(* CODESYS project MID_GPS_GPRS_Demo.project

Project tree, tasks and I/O mapping:
  Device : Changsha Xiangji-ARM Cortex A9(xilinx zynq7000)-linux, Changsha Xiangji Hiden Technology Co.Ltd, version 3.5.10.20
    application Application
      libraries: Standard, * (System); CAA DTUtil Extern, * (CAA Technical Workgroup); CAA SerialCom, * (CAA Technical Workgroup); CAA Types Extern, * (CAA Technical Workgroup); AC_Persistence, * (3S - Smart Software Solutions GmbH)
      task MainTask (cyclic, interval 4 ms, priority 1) calls MC20_serial, PLC_PRG
      task VISU_TASK (cyclic, interval 100 ms, priority 31) calls VisuElems.Visu_Prg
      program PLC_PRG [ST]
      global variables GVL
      program MC20_serial [ST]
      visualisation Main_test_Visua
    SoftMotion General Axis Pool
  text list GlobalTextList
*)

// Device/Application/GVL
{attribute 'qualified_only'}
{attribute 'qualified_only'}

VAR_GLOBAL

	NewDT : DT;
	NewDTS : STRING;
	NewDTSZH : STRING;
	cmdSend:BOOL := FALSE;
	recvOk:BOOL := FALSE;

	send_serial :BYTE := 0;

	
END_VAR

// Device/Application/MC20_serial
PROGRAM MC20_serial
VAR
	Com1Params: 			ARRAY [1..7] OF COM.PARAMETER;	(* Settings to communicate with the COM Port *)
	hCom: 					CAA.HANDLE;
	ComOpen: 				COM.Open;
	ComClose: 				COM.Close;
	ComWrite: 				COM.Write;
	ComRead: 				COM.Read;	
	//Writebuffer: 			STRING:= 'Hello! zhouqin';

	Snd_Cnt:				CAA.SIZE;

	Rcv_Cnt: 				CAA.SIZE;
	xCom1CloseError: 		BOOL;
	xCom1WriteError: 		BOOL;
	xCom1ReadError: 		BOOL;
	xError:					BOOL;
	
	uiComState: INT := 0;
	uiComState_MC20: INT := 0;
	ComID_MC20:USINT:=3;//串口号为4

	cmdSend:BOOL := FALSE;
	COMWritebufsum_MC20: 	    STRING(200):='';
	COMReadbufsum_MC20: 			STRING(200);
	ton2:TON;
	size:CAA.SIZE;
	
	at_ask_buffer1 :STRING(1000);
	at_ask_buffer2 :STRING(1000);
	at_ask_buffer3 :STRING(1000);
	at_ask_buffer4 :STRING(1000);
	at_ask_buffer5:STRING(1000);
	at_ask_buffer6 :STRING(1000);
	
	
	bit_start:INT;
	bit_end:INT;
	bit_start1:INT;
	bit_end1:INT;
	jd_info:STRING;
	wd_info:STRING;
	jd:REAL;
	wd:REAL;
	R_TIME:TIME;
	
END_VAR


CASE uiComState_MC20 OF
	0:
	Com1Params[1].udiParameterId := COM.CAA_Parameter_Constants.udiPort;
	Com1Params[1].udiValue := ComID_MC20; 
	Com1Params[2].udiParameterId := COM.CAA_Parameter_Constants.udiBaudrate;
	Com1Params[2].udiValue := 115200;
	Com1Params[3].udiParameterId := COM.CAA_Parameter_Constants.udiParity;
	Com1Params[3].udiValue := INT_TO_UINT(COM.PARITY.NONE);
	Com1Params[4].udiParameterId := COM.CAA_Parameter_Constants.udiStopBits;
	Com1Params[4].udiValue := INT_TO_UINT(COM.STOPBIT.ONESTOPBIT);
	Com1Params[5].udiParameterId := COM.CAA_Parameter_Constants.udiTimeout;
	Com1Params[5].udiValue := 0;
	Com1Params[6].udiParameterId := COM.CAA_Parameter_Constants.udiByteSize;
	Com1Params[6].udiValue := 8;
	Com1Params[7].udiParameterId := COM.CAA_Parameter_Constants.udiBinary;
	Com1Params[7].udiValue := 0;					
	ComOpen(xExecute := TRUE, usiListLength:=UINT_TO_USINT(SIZEOF(Com1Params)/SIZEOF(COM.PARAMETER)),pParameterList:= ADR(Com1Params),hCom=> hCom);			
	IF ComOpen.xError THEN
		uiComState_MC20 := 32767;
	ELSIF ComOpen.xDone THEN
		uiComState_MC20 := 1;
	END_IF
	
	1:
	COMWritebufsum_MC20:='AT$r';//发送AT指令，测试串口和MC20是否正常通信
	gvl.cmdSend:=TRUE;
	IF gvl.cmdSend  THEN
		ComWrite(xExecute := TRUE,hCom:= hCom,pBuffer:= ADR(COMWritebufsum_MC20),szSize:= ANY_TO_UDINT(len(COMWritebufsum_MC20)));		
		IF ComWrite.xError THEN
			uiComState_MC20 := 32767;
		END_IF
		IF ComWrite.xDone THEN		
			ComWrite(xExecute := FALSE);
			uiComState_MC20 := 2;
			gvl.send_serial := gvl.send_serial + 1;
			gvl.cmdSend := FALSE;
			gvl.recvOk := FALSE;
		END_IF
	END_IF
	
   2:
	TON2(IN:=TRUE,PT:=T#200MS);
		IF TON2.Q=TRUE THEN
	        	ComRead(xExecute := FALSE,hCom:= hCom, pBuffer:= ADR(COMReadbufsum_MC20), szBuffer:= SIZEOF(COMReadbufsum_MC20));	
	            COMReadbufsum_MC20:='';	
				uiComState_MC20 := 3;	
				TON2(IN:=FALSE,PT:=T#200MS);
		END_IF
	
	3:
	ComRead(xExecute := TRUE,hCom:= hCom, pBuffer:= ADR(COMReadbufsum_MC20), szBuffer:= SIZEOF(COMReadbufsum_MC20));
	IF ComRead.xError THEN
		uiComState_MC20 := 32767;
	END_IF	

    IF ComRead.xDone THEN
	  at_ask_buffer1:=COMReadbufsum_MC20;
	  uiComState_MC20 := 4;	
	END_IF


	4: 
	COMWritebufsum_MC20:='AT+QGNSSC=1$r';//发送AT指令，启动模块的GPS功能
	gvl.cmdSend:=TRUE;
	IF gvl.cmdSend  THEN
		ComWrite(xExecute := TRUE,hCom:= hCom,pBuffer:= ADR(COMWritebufsum_MC20),szSize:= ANY_TO_UDINT(len(COMWritebufsum_MC20)));		
		IF ComWrite.xError THEN
			uiComState_MC20 := 32767;
		END_IF
		IF ComWrite.xDone THEN		
			ComWrite(xExecute := FALSE);
			uiComState_MC20 := 5;
			gvl.send_serial := gvl.send_serial + 1;
			gvl.cmdSend := FALSE;
			gvl.recvOk := FALSE;
		END_IF
	END_IF
	
  5:
	TON2(IN:=TRUE,PT:=T#200MS);
		IF TON2.Q=TRUE THEN
                ComRead(xExecute := FALSE,hCom:= hCom, pBuffer:= ADR(COMReadbufsum_MC20), szBuffer:= SIZEOF(COMReadbufsum_MC20));		
	            COMReadbufsum_MC20:='';	
                uiComState_MC20 := 6;
				TON2(IN:=FALSE,PT:=T#200MS);
		END_IF
	
	6: 
	ComRead(xExecute := TRUE,hCom:= hCom, pBuffer:= ADR(COMReadbufsum_MC20), szBuffer:= SIZEOF(COMReadbufsum_MC20));
	IF ComRead.xError THEN
		uiComState_MC20 := 32767;
	END_IF

    IF ComRead.xDone THEN
	  at_ask_buffer2:=COMReadbufsum_MC20;
	  uiComState_MC20 := 7;	
	END_IF
	
	 7:

      uiComState_MC20 := 8;
	
	
	
	
	8:  
	COMWritebufsum_MC20:='AT+QGNSSRD="NMEA/RMC"$r';//发送AT指令，查询获取的经纬度
	gvl.cmdSend:=TRUE;
	IF gvl.cmdSend  THEN
		ComWrite(xExecute := TRUE,hCom:= hCom,pBuffer:= ADR(COMWritebufsum_MC20),szSize:= ANY_TO_UDINT(len(COMWritebufsum_MC20)));		
		IF ComWrite.xError THEN
			uiComState_MC20 := 32767;
		END_IF
		IF ComWrite.xDone THEN		
			ComWrite(xExecute := FALSE);
			uiComState_MC20 := 9;
			gvl.send_serial := gvl.send_serial + 1;
			gvl.cmdSend := FALSE;
			gvl.recvOk := FALSE;
		END_IF
	END_IF
	
	9:
	TON2(IN:=TRUE,PT:=T#200MS);
		IF TON2.Q=TRUE THEN
				ComRead(xExecute := FALSE,hCom:= hCom, pBuffer:= ADR(COMReadbufsum_MC20), szBuffer:= SIZEOF(COMReadbufsum_MC20));	//给xExecute制造一个上升沿，读串口命令才能被调用一次
	            COMReadbufsum_MC20:='';	
                uiComState_MC20 := 10;
				TON2(IN:=FALSE,PT:=T#200MS);
		END_IF
	
	10:
	ComRead(xExecute := TRUE,hCom:= hCom, pBuffer:= ADR(COMReadbufsum_MC20), szBuffer:= SIZEOF(COMReadbufsum_MC20));
	IF ComRead.xError THEN
		uiComState_MC20 := 32767;
	END_IF
    IF ComRead.xDone THEN
	  at_ask_buffer3:=COMReadbufsum_MC20;
	//解析经纬度信息，正确的 回复格式为消息：+QGNSSRD: $GNRMC,023740.000,A,2813.8648,N,11324.8867,E,0.42,353.49,020419,,,A*7C
   bit_start:=FIND( at_ask_buffer3,',A');
   bit_end:=FIND( at_ask_buffer3,',N');//读换行符的位置
   jd_info:=mid( at_ask_buffer3,bit_end-bit_start-1,bit_start+3);
   jd:=ANY_TO_REAL(jd_info)/100;
   bit_start1:=FIND( at_ask_buffer3,'N,');
   bit_end1:=FIND( at_ask_buffer3,',E');//读换行符的位置
   wd_info:=mid( at_ask_buffer3,bit_end1-bit_start1-1,bit_start1+2);
   wd:=ANY_TO_REAL(wd_info)/100;  
	 IF  jd=0 OR wd=0 THEN
		 uiComState_MC20 := 8;
     ELSE
		  uiComState_MC20 := 11;
	 END_IF
	  
	 	
	END_IF
	
	11:  
	COMWritebufsum_MC20:='AT+QNITZ=1$r';	//启用同步网络时间
	gvl.cmdSend:=TRUE;
	IF gvl.cmdSend  THEN
		ComWrite(xExecute := TRUE,hCom:= hCom,pBuffer:= ADR(COMWritebufsum_MC20),szSize:= ANY_TO_UDINT(len(COMWritebufsum_MC20)));		
		IF ComWrite.xError THEN
			uiComState_MC20 := 32767;
		END_IF
		IF ComWrite.xDone THEN		
			ComWrite(xExecute := FALSE);
			uiComState_MC20 := 12;
			gvl.send_serial := gvl.send_serial + 1;
			gvl.cmdSend := FALSE;
			gvl.recvOk := FALSE;
		END_IF
	END_IF
	
	12:
	TON2(IN:=TRUE,PT:=T#200MS);
		IF TON2.Q=TRUE THEN
				ComRead(xExecute := FALSE,hCom:= hCom, pBuffer:= ADR(COMReadbufsum_MC20), szBuffer:= SIZEOF(COMReadbufsum_MC20));	//给xExecute制造一个上升沿，读串口命令才能被调用一次
	            COMReadbufsum_MC20:='';	
                uiComState_MC20 := 13;
				TON2(IN:=FALSE,PT:=T#200MS);
		END_IF
	
	13:
	ComRead(xExecute := TRUE,hCom:= hCom, pBuffer:= ADR(COMReadbufsum_MC20), szBuffer:= SIZEOF(COMReadbufsum_MC20));
	IF ComRead.xError THEN
		uiComState_MC20 := 32767;
	END_IF
    IF ComRead.xDone THEN
	  at_ask_buffer4:=COMReadbufsum_MC20;
	  uiComState_MC20 := 14;	
	END_IF
	
    14:  
	COMWritebufsum_MC20:='AT+CCLK?$r';	//启获取模块的实时时钟
	gvl.cmdSend:=TRUE;
	IF gvl.cmdSend  THEN
		ComWrite(xExecute := TRUE,hCom:= hCom,pBuffer:= ADR(COMWritebufsum_MC20),szSize:= ANY_TO_UDINT(len(COMWritebufsum_MC20)));		
		IF ComWrite.xError THEN
			uiComState_MC20 := 32767;
		END_IF
		IF ComWrite.xDone THEN		
			ComWrite(xExecute := FALSE);
			uiComState_MC20 := 15;
			gvl.send_serial := gvl.send_serial + 1;
			gvl.cmdSend := FALSE;
			gvl.recvOk := FALSE;
		END_IF
	END_IF
	
	15:
	TON2(IN:=TRUE,PT:=T#200MS);
		IF TON2.Q=TRUE THEN
				ComRead(xExecute := FALSE,hCom:= hCom, pBuffer:= ADR(COMReadbufsum_MC20), szBuffer:= SIZEOF(COMReadbufsum_MC20));	//给xExecute制造一个上升沿，读串口命令才能被调用一次
	            COMReadbufsum_MC20:='';	
                uiComState_MC20 := 16;
				TON2(IN:=FALSE,PT:=T#200MS);
		END_IF
	
	16:
	ComRead(xExecute := TRUE,hCom:= hCom, pBuffer:= ADR(COMReadbufsum_MC20), szBuffer:= SIZEOF(COMReadbufsum_MC20));
	IF ComRead.xError THEN
		uiComState_MC20 := 32767;
	END_IF
    IF ComRead.xDone THEN
	  at_ask_buffer5:=COMReadbufsum_MC20;
      GVL.NewDTS:=MID(at_ask_buffer5,17,20);
	  
	  gvl.NewDTSZH:=CONCAT('DT#20',left(GVL.NewDTS,2));
	  gvl.NewDTSZH:=CONCAT(gvl.NewDTSZH,'-');	  
	  gvl.NewDTSZH:=CONCAT(gvl.NewDTSZH,mid(GVL.NewDTS,2,4));	 
      gvl.NewDTSZH:=CONCAT(gvl.NewDTSZH,'-');	
	  gvl.NewDTSZH:=CONCAT(gvl.NewDTSZH,mid(GVL.NewDTS,2,7));	
      gvl.NewDTSZH:=CONCAT(gvl.NewDTSZH,'-');	
 	  gvl.NewDTSZH:=CONCAT(gvl.NewDTSZH,mid(GVL.NewDTS,8,10));		  
	  GVL.NewDT:=ANY_TO_DT(gvl.NewDTSZH);
	  PLC_PRG.dtu_set_dt_fb.dtDateAndTime := STRING_TO_DT(gvl.NewDTSZH);
	  PLC_PRG.dtu_set_dt_fb(xExecute := FALSE);
	  PLC_PRG.dtu_set_dt_fb.xExecute := TRUE;
	  
	  
	  uiComState_MC20 := 32767;	
	END_IF
	255:
	
	32767:	
END_CASE

END_PROGRAM

// Device/Application/PLC_PRG
PROGRAM PLC_PRG
VAR
	ton1:TON;
	dtu_get_dt_fb:dtu.GetDateAndTime;
	Mydt:DT;
	MydtS:STRING;
END_VAR
VAR_INPUT	
	dtu_set_dt_fb: dtu.SetDateAndTime;
END_VAR



//时钟走时
    dtu_set_dt_fb();//将MC20读到的时钟同步到系统时钟里面去
	TON1(IN:=TRUE,PT:=T#1S);//系统时钟走时，每秒读一次系统时钟
		IF TON1.Q=TRUE THEN
				Mydt:=GETdatetime();		
				MydtS:=ANY_TO_STRING(Mydt);
				TON1(IN:=FALSE,PT:=T#1S);
		END_IF

END_PROGRAM

// Device/Application/Main_test_Visua
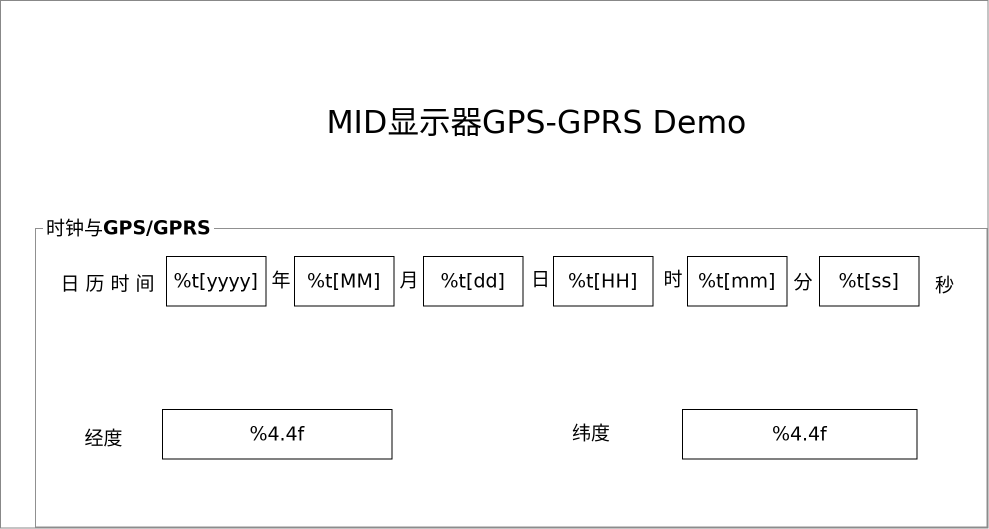
VISUALIZATION Main_test_Visua  // 989x529
    GroupBox (35,220 952x307), "时钟与GPS/GPRS"
        Rectangle (127,189 230x50), "%4.4f", text variable: MC20_serial.jd
        Rectangle (647,189 235x50), "%4.4f", text variable: MC20_serial.wd
        Label (507,186 98x54), "纬度"
        Label (12,188 113x60), "经度"
        Rectangle (784,36 100x50), "%t[ss]", text variable: PLC_PRG.MydtS
        Label (742,29 52x66), "分"
        Rectangle (652,36 100x50), "%t[mm]", text variable: PLC_PRG.MydtS
        Label (607,26 62x66), "时"
        Label (473,25 65x68), "日"
        Label (219,25 54x70), "年"
        Label (343,23 62x74), "月"
        Rectangle (518,36 100x50), "%t[HH]", text variable: PLC_PRG.MydtS
        Rectangle (388,36 100x50), "%t[dd]", text variable: PLC_PRG.MydtS
        Rectangle (259,36 100x50), "%t[MM]", text variable: PLC_PRG.MydtS
        Rectangle (131,36 100x50), "%t[yyyy]", text variable: PLC_PRG.MydtS
        Label (2,32 141x63), "日 历 时 间"
        Label (876,34 67x62), "秒"
    Label (250,79 574x86), "MID显示器GPS-GPRS Demo"
END_VISUALIZATION
